FUNCTION_BLOCK FB_GetCPULoadPLC
VAR_INPUT
	rInterval			: REAL := 10.0;		// [sec]
END_VAR
VAR_OUTPUT
	rCPULoad			: REAL;				// [deg]
	bError				: BOOL;				// error flag (indicator: error occured)
	nErrID				: UDINT;			// last error ID 
END_VAR
VAR
	// internal use
	sAmsNetId			: T_AmsNetId;		// ADS Net ID (local = '')    
	iState				: INT;
	// FB instances
	fbReadCPUUsage		: TC_CpuUsage;  
	tonInterval			: Tc2_Standard.TON;
	// Info
	iErrorCnt			: UINT;
	iGoodCnt			: UINT;
END_VAR


// Interval timer
tonInterval(IN := NOT tonInterval.Q, PT := REAL_TO_TIME(rInterval * 1000.0));

CASE iState OF
	0: // Initiate program parameters (if required)
		fbReadCPUUsage(START := FALSE);
		IF (tonInterval.Q) THEN
			iState := 10;
		END_IF

	10:	// Trigger FB: request CPU data
		fbReadCPUUsage(	NETID := sAmsNetId,
						START := TRUE,
						TMOUT := T#5S	);
		IF (fbReadCPUUsage.BUSY) THEN
			// Started
			iState := 20;
		ELSIF (fbReadCPUUsage.ERR) THEN
			// Error
			iErrorCnt := iErrorCnt + 1;
			iState := 0;
		END_IF

	20:	// Process FB: Request CPU temp
		fbReadCPUUsage(START := FALSE); 
		IF (NOT fbReadCPUUsage.BUSY) THEN
			IF (NOT fbReadCPUUsage.ERR) THEN
				rCPULoad := fbReadCPUUsage.USAGE;
				iGoodCnt := iGoodCnt + 1;
				iState := 30;
			ELSE
				iErrorCnt := iErrorCnt + 1;
				iState := 0;
			END_IF                                               
		END_IF
    
     30: // Done 
		iState := 0;

	ELSE
		iState := 0; 

END_CASE

bError := fbReadCPUUsage.ERR;
nErrID := fbReadCPUUsage.ERRID;

END_FUNCTION_BLOCK

(* stored: Version 1.1.0.1, ProductVersion 3.1.4024.5
   POU FB_GetCPULoadPLC: Id {c3fd5c4f-fb3a-4210-bfd4-7cf02d7d0e7e}, SpecialFunc None *)
